(* PLC project LD_EVOLUTION_2, Beckhoff Automation GmbH TwinCAT PLC Control 3.5.10.30 *)
(* stored: creationDateTime 2019-09-26T16:14:26.3083942, modificationDateTime 2019-09-26T16:14:26.3083942 *)

PROGRAM Main
VAR
	A: BOOL;
	B: BOOL;
	Open: BOOL;
	C: BOOL;
END_VAR

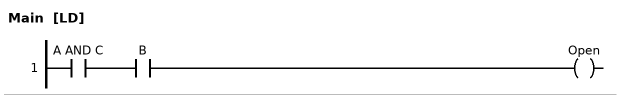
(* LD diagram, written out as Structured Text *)

Open := (A AND C) AND B;
END_PROGRAM

CONFIGURATION Application
  RESOURCE LD_EVOLUTION_2 ON PLC
    TASK PlcTask(INTERVAL := T#0ms, PRIORITY := 20);
    PROGRAM Main WITH PlcTask : Main;
  END_RESOURCE
END_CONFIGURATION
